FUNCTION_BLOCK FB_GeneratorEX EXTENDS FB_Generator
VAR_INPUT
END_VAR
VAR_OUTPUT
END_VAR
VAR
END_VAR

METHOD Flash : BOOL
VAR_INPUT
END_VAR
fbTon1(IN:=NOT fbTon1.Q , PT:= 2* tCycletime , Q=> , ET=> );
Flash := fbTon1.ET < fbTon1.PT / 3;
END_METHOD

PROPERTY Vendor : STRING
GET
Vendor := CONCAT
			(
			STR1:= 'Company b, based on' , 
			STR2:=SUPER^.Vendor 
			);
END_GET
END_PROPERTY

END_FUNCTION_BLOCK

(* stored: Version 1.1.0.1, ProductVersion 3.1.4024.6
   POU FB_GeneratorEX: Id {9012c853-6432-4b40-abf2-3588accf353e}, SpecialFunc None
   Method Flash: Id {40f36b06-d4fe-448d-98f3-dcf1fbe0ed04}
   Property Vendor: Id {8c577059-e7b8-4609-8064-3f92451d9660}
   Get Get: Id {76c9f737-cae0-4a2e-9dfc-925662454ae9} *)
